// TIA Portal V19 export
FUNCTION "Set_Pop_Up_Blocking" : Void   // FC36, STL
TITLE = Send start blocking pop up text to intouch PC
{ S7_Optimized_Access := 'TRUE' }
AUTHOR : FLA
FAMILY : UHT
VERSION : 1.0
// Text number must be loaded in to ACC 1 before calling FC36
// 
// Max number off intouch PC's = 8
// 
// FC 36 using DB 36
// 
// FC 37 reset all text numbers after 5 seconds
// 
// Programmer Init: 8953-FLA
// 
// Change Log:
// 
// Date        Change                          Updated by
// ------------------------------------------------------
// 19.04.99    1. Edition                      FLA
// stored: AutoNumber false
   VAR_INPUT
      alarmTextNum : Int;
   END_VAR
BEGIN

NETWORK
TITLE = 
// pop up text number from program in ACC 1
//    OPN   "PopUpBitToScada"    // Command from intouch pc number x ( 1 - 8 )
      L     "PopUpBitToScada".PC_number_from_intouch;  // jump to pc number X
      JL    M001;  //
      JU    M002;  // if PC 0
      JU    M003;  // if PC 1
      JU    M004;  // if PC 2
      JU    M005;  // if PC 3
      JU    M006;  // if PC 4
      JU    M007;  // if PC 5
      JU    M008;  // if PC 6
      JU    M009;  // if PC 7
      JU    M00a;  // if PC 8
M001: JU    M002;  // if PC 9


M003: L     #alarmTextNum;
      T     "PopUpBitToScada".Pop_up_text_to_PC1;  // Send text to PC 1
      JU    M00b;  // jump to ok and reset pc number

M004: L     #alarmTextNum;
      T     "PopUpBitToScada".Pop_up_text_to_PC2;  // Send text to PC 1
      JU    M00b;  // jump to ok and reset pc number

M005: L     #alarmTextNum;
      T     "PopUpBitToScada".Pop_up_text_to_PC3;  // Send text to PC 1
      JU    M00b;  // jump to ok and reset pc number

M006: L     #alarmTextNum;
      T     "PopUpBitToScada".Pop_up_text_to_PC4;  // Send text to PC 1
      JU    M00b;  // jump to ok and reset pc number

M007: L     #alarmTextNum;
      T     "PopUpBitToScada".Pop_up_text_to_PC5;  // Send text to PC 1
      JU    M00b;  // jump to ok and reset pc number

M008: L     #alarmTextNum;
      T     "PopUpBitToScada".Pop_up_text_to_PC6;  // Send text to PC 1
      JU    M00b;  // jump to ok and reset pc number

M009: L     #alarmTextNum;
      T     "PopUpBitToScada".Pop_up_text_to_PC7;  // Send text to PC 1
      JU    M00b;  // jump to ok and reset pc number

M00a: L     #alarmTextNum;
      T     "PopUpBitToScada".Pop_up_text_to_PC8;  // Send text to PC 1
      JU    M00b;  // jump to ok and reset pc number

M00b: L     0;
      T     "PopUpBitToScada".PC_number_from_intouch;  //Send text to PC 9
      L     5;
      T     "PopUpBitToScada".Count_down_to_reset;

M002: NOP   0;  // Reset PC number
END_FUNCTION
